% RSLogix 500 project P2_22_BAK013.RSS, saved by version 8.30.00.16 %
PROJECT "UNTITLED"    % processor: Bul.1763 MicroLogix 1100 Series B %

PROGRAM FILES
  LAD 2   4 rungs
  LAD 3 "I/O"  8 rungs
  LAD 4 "CTRL"  6 rungs
  LAD 5 "CYCLE"  5 rungs

DATA FILES
  O0 OUTPUT  4 elements
  I1 INPUT  6 elements
  S2 STATUS  66 elements
  B3 BINARY  1 elements
  T4 TIMER  1 elements
  C5 COUNTER  1 elements
  R6 CONTROL  1 elements
  N7 INTEGER  1 elements
  F8 FLOAT  1 elements

LADDER 2
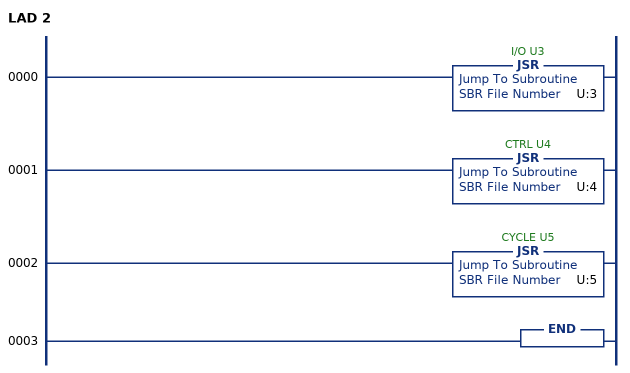
% Rung: 0 %
SOR JSR U:3 EOR
%   U:3  U3  "I/O" %
% Rung: 1 %
SOR JSR U:4 EOR
%   U:4  U4  "CTRL" %
% Rung: 2 %
SOR JSR U:5 EOR
%   U:5  U5  "CYCLE" %
% Rung: 3 %
SOR END EOR

LADDER 3 "I/O"
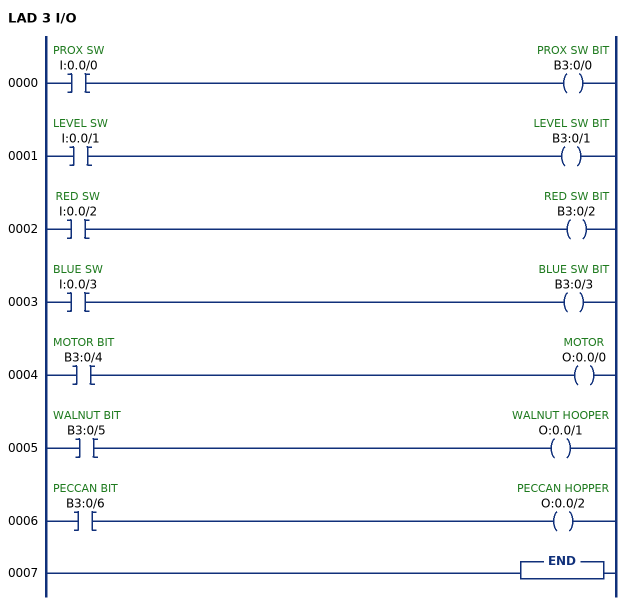
% Rung: 0 %
SOR XIC I:0.0/0 OTE B3:0/0 EOR
%   I:0.0/0  "PROX SW" %
%   B3:0/0  "PROX SW BIT" %
% Rung: 1 %
SOR XIC I:0.0/1 OTE B3:0/1 EOR
%   I:0.0/1  "LEVEL SW" %
%   B3:0/1  "LEVEL SW BIT" %
% Rung: 2 %
SOR XIC I:0.0/2 OTE B3:0/2 EOR
%   I:0.0/2  "RED SW" %
%   B3:0/2  "RED SW BIT" %
% Rung: 3 %
SOR XIC I:0.0/3 OTE B3:0/3 EOR
%   I:0.0/3  "BLUE SW" %
%   B3:0/3  "BLUE SW BIT" %
% Rung: 4 %
SOR XIC B3:0/4 OTE O:0.0/0 EOR
%   B3:0/4  "MOTOR BIT" %
%   O:0.0/0  "MOTOR" %
% Rung: 5 %
SOR XIC B3:0/5 OTE O:0.0/1 EOR
%   B3:0/5  "WALNUT BIT" %
%   O:0.0/1  "WALNUT HOOPER" %
% Rung: 6 %
SOR XIC B3:0/6 OTE O:0.0/2 EOR
%   B3:0/6  "PECCAN BIT" %
%   O:0.0/2  "PECCAN HOPPER" %
% Rung: 7 %
SOR END EOR

LADDER 4 "CTRL"
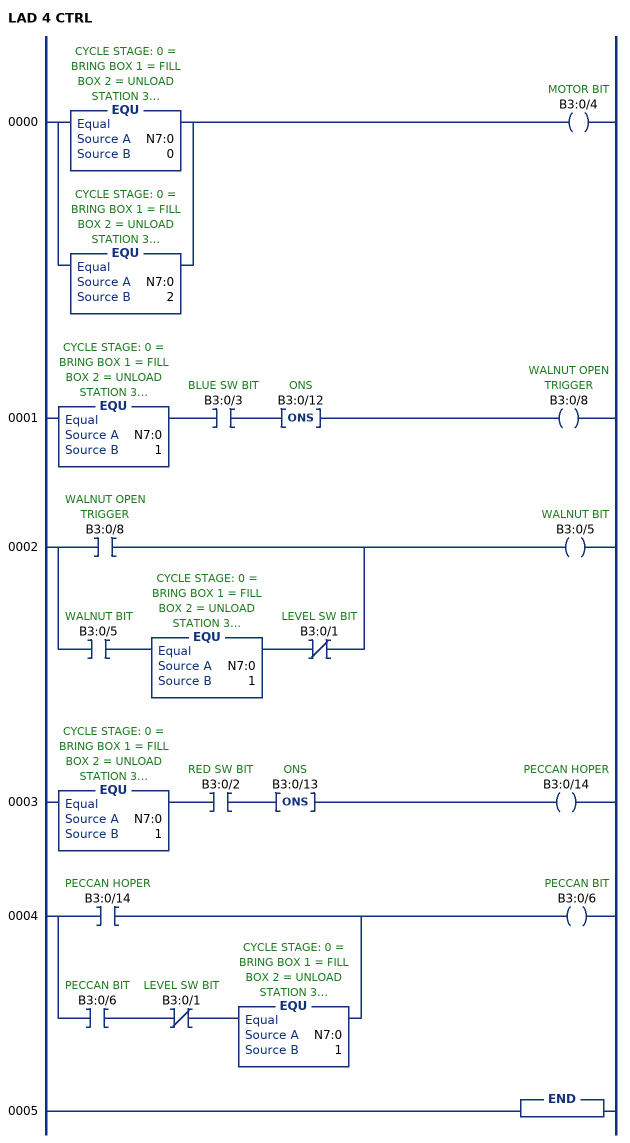
% Rung: 0 %
SOR BST EQU N7:0 0 NXB EQU N7:0 2 BND OTE B3:0/4 EOR
%   N7:0  "CYCLE STAGE: 0 = BRING BOX 1 = FILL BOX 2 = UNLOAD STATION 3= INTERMEDIATE" %
%   B3:0/4  "MOTOR BIT" %
% Rung: 1 %
SOR EQU N7:0 1 XIC B3:0/3 ONS B3:0/12 OTE B3:0/8 EOR
%   N7:0  "CYCLE STAGE: 0 = BRING BOX 1 = FILL BOX 2 = UNLOAD STATION 3= INTERMEDIATE" %
%   B3:0/3  "BLUE SW BIT" %
%   B3:0/12  "ONS" %
%   B3:0/8  "WALNUT OPEN TRIGGER" %
% Rung: 2 %
SOR BST XIC B3:0/8 NXB XIC B3:0/5 EQU N7:0 1 XIO B3:0/1 BND OTE B3:0/5 EOR
%   B3:0/8  "WALNUT OPEN TRIGGER" %
%   B3:0/5  "WALNUT BIT" %
%   N7:0  "CYCLE STAGE: 0 = BRING BOX 1 = FILL BOX 2 = UNLOAD STATION 3= INTERMEDIATE" %
%   B3:0/1  "LEVEL SW BIT" %
% Rung: 3 %
SOR EQU N7:0 1 XIC B3:0/2 ONS B3:0/13 OTE B3:0/14 EOR
%   N7:0  "CYCLE STAGE: 0 = BRING BOX 1 = FILL BOX 2 = UNLOAD STATION 3= INTERMEDIATE" %
%   B3:0/2  "RED SW BIT" %
%   B3:0/13  "ONS" %
%   B3:0/14  "PECCAN HOPER" %
% Rung: 4 %
SOR BST XIC B3:0/14 NXB XIC B3:0/6 XIO B3:0/1 EQU N7:0 1 BND OTE B3:0/6 EOR
%   B3:0/14  "PECCAN HOPER" %
%   B3:0/6  "PECCAN BIT" %
%   B3:0/1  "LEVEL SW BIT" %
%   N7:0  "CYCLE STAGE: 0 = BRING BOX 1 = FILL BOX 2 = UNLOAD STATION 3= INTERMEDIATE" %
% Rung: 5 %
SOR END EOR

LADDER 5 "CYCLE"
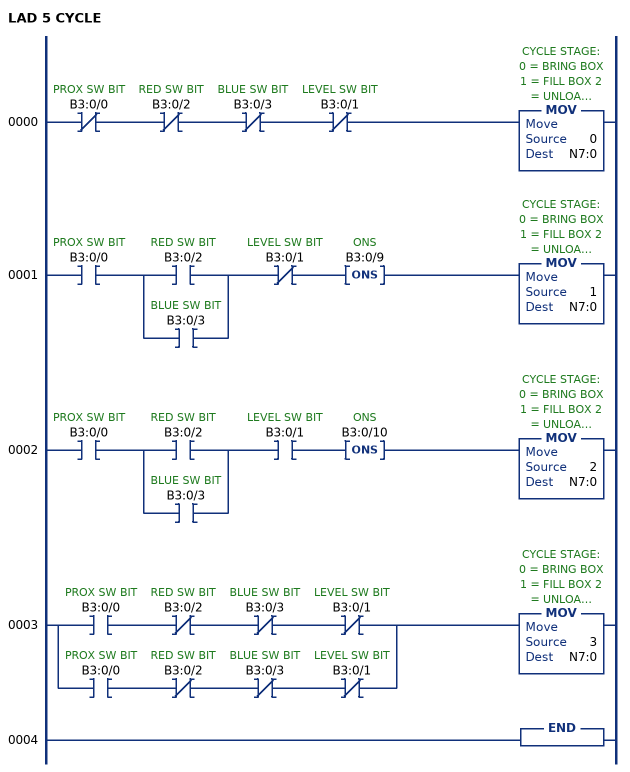
% Rung: 0 %
SOR XIO B3:0/0 XIO B3:0/2 XIO B3:0/3 XIO B3:0/1 MOV 0 N7:0 EOR
%   B3:0/0  "PROX SW BIT" %
%   B3:0/2  "RED SW BIT" %
%   B3:0/3  "BLUE SW BIT" %
%   B3:0/1  "LEVEL SW BIT" %
%   N7:0  "CYCLE STAGE: 0 = BRING BOX 1 = FILL BOX 2 = UNLOAD STATION 3= INTERMEDIATE" %
% Rung: 1 %
SOR XIC B3:0/0 BST XIC B3:0/2 NXB XIC B3:0/3 BND XIO B3:0/1 ONS B3:0/9 MOV 1 N7:0 EOR
%   B3:0/0  "PROX SW BIT" %
%   B3:0/2  "RED SW BIT" %
%   B3:0/3  "BLUE SW BIT" %
%   B3:0/1  "LEVEL SW BIT" %
%   B3:0/9  "ONS" %
%   N7:0  "CYCLE STAGE: 0 = BRING BOX 1 = FILL BOX 2 = UNLOAD STATION 3= INTERMEDIATE" %
% Rung: 2 %
SOR XIC B3:0/0 BST XIC B3:0/2 NXB XIC B3:0/3 BND XIC B3:0/1 ONS B3:0/10 MOV 2 N7:0 EOR
%   B3:0/0  "PROX SW BIT" %
%   B3:0/2  "RED SW BIT" %
%   B3:0/3  "BLUE SW BIT" %
%   B3:0/1  "LEVEL SW BIT" %
%   B3:0/10  "ONS" %
%   N7:0  "CYCLE STAGE: 0 = BRING BOX 1 = FILL BOX 2 = UNLOAD STATION 3= INTERMEDIATE" %
% Rung: 3 %
SOR BST XIC B3:0/0 XIO B3:0/2 XIO B3:0/3 XIO B3:0/1 NXB XIC B3:0/0 XIO B3:0/2 XIO B3:0/3 XIO B3:0/1 BND MOV 3 N7:0 EOR
%   B3:0/0  "PROX SW BIT" %
%   B3:0/2  "RED SW BIT" %
%   B3:0/3  "BLUE SW BIT" %
%   B3:0/1  "LEVEL SW BIT" %
%   N7:0  "CYCLE STAGE: 0 = BRING BOX 1 = FILL BOX 2 = UNLOAD STATION 3= INTERMEDIATE" %
% Rung: 4 %
SOR END EOR

DATA TABLE (non-zero values as saved)
DATA B3
% B3:0 % 0X2200
